FUNCTION_BLOCK FB_Pusher_Itf
VAR_INPUT
	i_ifRegister : IF_Register;
	
END_VAR
VAR_OUTPUT
END_VAR
VAR
	diProductCounter : DINT;
	ifFillRegister : IF_FillRegister;
	
	xSucess: BOOL;
END_VAR

VAR_IN_OUT
	iq_xSensor: BOOL;
END_VAR

xSucess :=__QUERYINTERFACE(i_ifRegister,ifFillRegister);
IF xSucess THEN
	diProductCounter := diProductCounter+1;
	IF iq_xSensor AND ifFillRegister.xReadyForPut THEN
		iq_xSensor:=FALSE;
		ifFillRegister.put(i_diInValue:=diProductCounter);
	END_IF
END_IF

END_FUNCTION_BLOCK

(* stored: Version 1.1.0.1
   POU FB_Pusher_Itf: Id {6a404b73-fb82-4d5a-a295-ca4edb8c2080}, SpecialFunc None *)
